// TwinCAT 3 PLC project PLC
// ProgramVersion: 3.1.4024.0
// libraries:
//   Tc2_Standard, * (Beckhoff Automation GmbH)
//   Tc2_System, * (Beckhoff Automation GmbH)
//   Tc2_Utilities, * (Beckhoff Automation GmbH)
//   Tc3_IotBase, * (Beckhoff Automation GmbH)
//   Tc3_IotCommunicator, * (Beckhoff Automation GmbH)
//   Tc3_Module, * (Beckhoff Automation GmbH)
// project tree:
//   00_HMI/DUTs/ ST_HMI_Variable_Mapping.TcDUT, ST_IoT_Device_General.TcDUT
//   00_HMI/DUTs/Widgets/ ST_IoT_HMI_General_Widget.TcDUT, ST_IoT_HMI_General_Widget_Plug.TcDUT, ST_IoT_HMI_General_Widget_RGBW.TcDUT, ST_IoT_HMI_General_Widget_Timer.TcDUT
//   DUTs/ProjectSpecific/HMI/00_Home/ ST_IoT_HMI_Rooms.TcDUT
//   DUTs/ProjectSpecific/HMI/100_FirstFloor/110_Entrance/ ST_IoT_HMI_Entrance.TcDUT
//   DUTs/ProjectSpecific/HMI/100_FirstFloor/120_Toilette/ ST_IoT_HMI_Toilette.TcDUT
//   DUTs/ProjectSpecific/HMI/100_FirstFloor/130_LivingRoom/ ST_IoT_HMI_LivingRoom.TcDUT
//   DUTs/ProjectSpecific/HMI/100_FirstFloor/140_Kitchen/ ST_IoT_HMI_Kitchen.TcDUT
//   DUTs/ProjectSpecific/HMI/100_FirstFloor/150_Storage/ ST_IoT_HMI_Storage.TcDUT
//   DUTs/ProjectSpecific/HMI/200_SecondFloor/210_Stairs/ ST_IoT_HMI_Stairs.TcDUT
//   DUTs/ProjectSpecific/HMI/200_SecondFloor/220_Office/ ST_IoT_HMI_Office.TcDUT
//   DUTs/ProjectSpecific/HMI/200_SecondFloor/230_Bathroom/ ST_IoT_HMI_Bathroom.TcDUT
//   DUTs/ProjectSpecific/HMI/200_SecondFloor/240_Bedroom/ ST_IoT_HMI_Bedroom.TcDUT
//   DUTs/ProjectSpecific/Rooms/Devices/ ST_Esp32_BedLight.TcDUT, ST_StatusDevices.TcDUT, ST_StatusShellyOnePM.TcDUT
//   DUTs/ProjectSpecific/Rooms/ ST_BedroomDevices.TcDUT, ST_LivingRoomDevices.TcDUT
//   / FC_MemcpyLimited.TcPOU, PlcTask.TcTTO
//   GVLs/ GVL_HMI.TcGVL, GVL_Devices.TcGVL
//   00_MQTT/DUT/ ST_MqttClient.TcDUT, ST_MqttConfig.TcDUT, ST_MqttData.TcDUT
//   00_MQTT/GVL/ GVL_Mqtt.TcGVL
//   POUs/00_HMI_Connection/ FB_IoT_HMI_Connection.TcPOU, PRG_IoT_HMI_Connection.TcPOU
//   POUs/00_MQTT_Connection/ FB_IoT_MqttClient.TcPOU
//   POUs/130_LivingRoom/ FB_LivingRoom.TcPOU, PRG_LivingRoom.TcPOU
//   POUs/ MAIN.TcPOU
// real-time tasks:
//   TASK PlcTask: cycle T#10ms, priority 6, ADS port 350

CONFIGURATION PLC
    RESOURCE PLC ON TwinCAT3
        TASK PlcTask(INTERVAL := T#10ms, PRIORITY := 6);
        PROGRAM MAIN WITH PlcTask : MAIN;
    END_RESOURCE
END_CONFIGURATION

// ---- 00_HMI/DUTs/ST_HMI_Variable_Mapping.TcDUT
TYPE ST_HMI_Variable_Mapping :
STRUCT
	sPath					: BOOL;
	
END_STRUCT
END_TYPE

// ---- 00_HMI/DUTs/ST_IoT_Device_General.TcDUT
TYPE ST_IoT_Device_General :
STRUCT

	sDeviceName					: STRING;	
	sDeviceIcon					: STRING;
	sMainTopic					: STRING;
	
END_STRUCT
END_TYPE

// ---- 00_HMI/DUTs/Widgets/ST_IoT_HMI_General_Widget.TcDUT
TYPE ST_IoT_HMI_General_Widget :
STRUCT
	sDisplayName 				: STRING := '';
	bValue1 					: BOOL := FALSE;
	{attribute 'iot.Unit' := '%'}
	{attribute 'iot.MinValue' := '0'}
	{attribute 'iot.MaxValue' := '100'}
	nValue2 					: INT;
	nValue2Request 				: INT;
	bValue2Up 					: BOOL;
	bValue2Down 				: BOOL;
	{attribute 'iot.Unit' := '%'}
	{attribute 'iot.MinValue' := '0'}
	{attribute 'iot.MaxValue' := '100'}
	nValue3 					: INT;
	nValue3Request 				: INT;
	bValue3Up 					: BOOL;
	bValue3Down 				: BOOL;
	sMode1 						: STRING := 'Automatic';
	aModes1 					: ARRAY[0..1] OF STRING := ['Manual', 'Automatic'];
	sMode2 						: STRING := 'Automatic';
	aModes2 					: ARRAY[0..2] OF STRING := ['Manual', 'Automatic', 'Next Mode'];
	sMode3 						: STRING := 'Automatic';
	aModes3 					: ARRAY[0..1] OF STRING := ['Manual', 'Automatic'];
END_STRUCT
END_TYPE

// ---- 00_HMI/DUTs/Widgets/ST_IoT_HMI_General_Widget_Plug.TcDUT
TYPE ST_IoT_HMI_General_Widget_Plug :
STRUCT
	
	sDisplayName 					: STRING := 'Plug';
	bOn 							: BOOL;
	sMode 							: STRING := 'Automatic';
	aModes 							: ARRAY[0..1] OF STRING := ['Manual', 'Automatic'];
	
END_STRUCT
END_TYPE

// ---- 00_HMI/DUTs/Widgets/ST_IoT_HMI_General_Widget_RGBW.TcDUT
TYPE ST_IoT_HMI_General_Widget_RGBW :
STRUCT
	sDisplayName 						: STRING := '';
	bLight 								: BOOL := FALSE;
	{attribute 'iot.Unit' := '%'}
	{attribute 'iot.MinValue' := '0'}
	{attribute 'iot.MaxValue' := '100'}
	nLight 								: INT := 100;
	nHueValue 							: INT := 57;
	nSaturation 						: INT := 100;
	{attribute 'iot.MinValue' := '2400'} 
	{attribute 'iot.MaxValue' := '6500'}
	nColorTemperature 					: INT := 3500;
	sMode 								: STRING := 'Permanent';
	aModes 								: ARRAY[0..4] OF STRING := ['Permanent', '15 Minuten', '30 Minuten', '45 Minuten', '1 Stunde'];
END_STRUCT
END_TYPE

// ---- 00_HMI/DUTs/Widgets/ST_IoT_HMI_General_Widget_Timer.TcDUT
TYPE ST_IoT_HMI_General_Widget_Timer :
STRUCT
	bLight			: BOOL;
	{attribute 'iot.Unit':='min'}
	{attribute 'iot.MinValue':='0'}
	{attribute 'iot.MaxValue':='120'}
	nLight			: INT;	
	sMode			: STRING;
	aModes			: ARRAY[0..1] OF STRING;
END_STRUCT
END_TYPE

// ---- DUTs/ProjectSpecific/HMI/00_Home/ST_IoT_HMI_Rooms.TcDUT
TYPE ST_IoT_HMI_Rooms :
STRUCT
	
	// First floor
	{attribute 'iot.DisplayName' := 'Flur UG'}
	{attribute 'iot.NestedStructIcon' := 'Door_Open'}
	sEntrance					: ST_IoT_HMI_Entrance;	
	{attribute 'iot.DisplayName' := 'Toilette'}
	{attribute 'iot.NestedStructIcon' := 'Toilet'}
	sToilette					: ST_IoT_HMI_Toilette;
	{attribute 'iot.DisplayName' := 'Wohnzimmer'}
	{attribute 'iot.NestedStructIcon' := 'Sofa'}
	sLivingRoom					: ST_IoT_HMI_LivingRoom;
	{attribute 'iot.DisplayName' := 'Kueche'}
	{attribute 'iot.NestedStructIcon' := 'Kitchen'}
	sKitchen					: ST_IoT_HMI_Kitchen;
	{attribute 'iot.DisplayName' := 'Speiss'}
	{attribute 'iot.NestedStructIcon' := 'Storage'}
	sStorage					: ST_IoT_HMI_Storage;
	
	// Second floor
	{attribute 'iot.DisplayName' := 'Flur OG'}
	{attribute 'iot.NestedStructIcon' := 'Floor'}
	sStairs						: ST_IoT_HMI_Stairs;
	{attribute 'iot.DisplayName' := 'Buero'}
	{attribute 'iot.NestedStructIcon' := 'PC'}
	sOffice						: ST_IoT_HMI_Office;
	{attribute 'iot.DisplayName' := 'Badezimmer'}
	{attribute 'iot.NestedStructIcon' := 'Bath'}
	sBathroom					: ST_IoT_HMI_Bathroom;
	{attribute 'iot.DisplayName' := 'Schlafzimmer'}
	{attribute 'iot.NestedStructIcon' := 'Bed'}
	sBedroom					: ST_IoT_HMI_Bedroom;
	
END_STRUCT
END_TYPE

// ---- DUTs/ProjectSpecific/HMI/100_FirstFloor/110_Entrance/ST_IoT_HMI_Entrance.TcDUT
TYPE ST_IoT_HMI_Entrance :
STRUCT
	
	{attribute 'iot.ReadOnly' := 'false'}
	{attribute 'iot.DisplayName' := 'Light'}
	{attribute 'iot.WidgetType' := 'General'}
	{attribute 'iot.GeneralWidgetIcon' := 'Lightbulb'}
	{attribute 'iot.GeneralWidgetColor' := 'LightSlateGray'}
	{attribute 'iot.GeneralValue1SwitchVisible' := 'true'}
	{attribute 'iot.GeneralValue2Visible' := 'false'}
	{attribute 'iot.GeneralValue2SliderVisible' := 'false'}
	{attribute 'iot.GeneralValue2SliderValuesVisible' := 'false'}
	{attribute 'iot.GeneralValue2SliderButtonsVisible' := 'false'}
	{attribute 'iot.GeneralValue2SliderButtonsInverted' := 'false'}
	{attribute 'iot.GeneralValue3Visible' := 'false'}
	{attribute 'iot.GeneralValue3SliderVisible' := 'false'}
	{attribute 'iot.GeneralValue3SliderValuesVisible' := 'false'}
	{attribute 'iot.GeneralValue3SliderButtonsVisible' := 'false'}
	{attribute 'iot.GeneralValue3SliderButtonsInverted' := 'false'}
	{attribute 'iot.GeneralMode1Visible' := 'false'}
	{attribute 'iot.GeneralMode1Changeable' := 'false'}
	{attribute 'iot.GeneralMode2Visible' := 'false'}
	{attribute 'iot.GeneralMode2Changeable' := 'false'}
	{attribute 'iot.GeneralMode3Visible' := 'false'}
	{attribute 'iot.GeneralMode3Changeable' := 'false'}
	sLight						: ST_IoT_HMI_General_Widget;
    
	{attribute 'iot.ReadOnly' := 'false'}
	{attribute 'iot.DisplayName' := 'Steckdose'}
	{attribute 'iot.WidgetType' := 'Plug'}
	{attribute 'iot.PlugModeVisible' := 'true'}
	{attribute 'iot.PlugModeChangeable' := 'true'}
	sPlug					 	: ST_IoT_HMI_General_Widget_Plug;		

END_STRUCT
END_TYPE

// ---- DUTs/ProjectSpecific/HMI/100_FirstFloor/120_Toilette/ST_IoT_HMI_Toilette.TcDUT
TYPE ST_IoT_HMI_Toilette :
STRUCT
	
	{attribute 'iot.ReadOnly' := 'false'}
	{attribute 'iot.DisplayName' := 'Light'}
	{attribute 'iot.WidgetType' := 'General'}
	{attribute 'iot.GeneralWidgetIcon' := 'Lightbulb'}
	{attribute 'iot.GeneralWidgetColor' := 'FF00BFFF'}
	{attribute 'iot.GeneralValue1SwitchVisible' := 'true'}
	{attribute 'iot.GeneralValue2Visible' := 'false'}
	{attribute 'iot.GeneralValue2SliderVisible' := 'false'}
	{attribute 'iot.GeneralValue2SliderValuesVisible' := 'false'}
	{attribute 'iot.GeneralValue2SliderButtonsVisible' := 'false'}
	{attribute 'iot.GeneralValue2SliderButtonsInverted' := 'false'}
	{attribute 'iot.GeneralValue3Visible' := 'false'}
	{attribute 'iot.GeneralValue3SliderVisible' := 'false'}
	{attribute 'iot.GeneralValue3SliderValuesVisible' := 'false'}
	{attribute 'iot.GeneralValue3SliderButtonsVisible' := 'false'}
	{attribute 'iot.GeneralValue3SliderButtonsInverted' := 'false'}
	{attribute 'iot.GeneralMode1Visible' := 'false'}
	{attribute 'iot.GeneralMode1Changeable' := 'false'}
	{attribute 'iot.GeneralMode2Visible' := 'false'}
	{attribute 'iot.GeneralMode2Changeable' := 'false'}
	{attribute 'iot.GeneralMode3Visible' := 'false'}
	{attribute 'iot.GeneralMode3Changeable' := 'false'}
	sLight						: ST_IoT_HMI_General_Widget;
    
	{attribute 'iot.ReadOnly' := 'false'}
	{attribute 'iot.DisplayName' := 'Steckdose'}
	{attribute 'iot.WidgetType' := 'Plug'}
	{attribute 'iot.PlugModeVisible' := 'true'}
	{attribute 'iot.PlugModeChangeable' := 'true'}
	sPlug					 	: ST_IoT_HMI_General_Widget_Plug;	

END_STRUCT
END_TYPE

// ---- DUTs/ProjectSpecific/HMI/100_FirstFloor/130_LivingRoom/ST_IoT_HMI_LivingRoom.TcDUT
TYPE ST_IoT_HMI_LivingRoom :
STRUCT
	
	{attribute 'iot.ReadOnly' := 'false'}
	{attribute 'iot.DisplayName' := 'Light'}
	{attribute 'iot.WidgetType' := 'General'}
	{attribute 'iot.GeneralWidgetIcon' := 'Lightbulb'}
	{attribute 'iot.GeneralWidgetColor' := 'FF00BFFF'}
	{attribute 'iot.GeneralValue1SwitchVisible' := 'true'}
	{attribute 'iot.GeneralValue2Visible' := 'false'}
	{attribute 'iot.GeneralValue2SliderVisible' := 'false'}
	{attribute 'iot.GeneralValue2SliderValuesVisible' := 'false'}
	{attribute 'iot.GeneralValue2SliderButtonsVisible' := 'false'}
	{attribute 'iot.GeneralValue2SliderButtonsInverted' := 'false'}
	{attribute 'iot.GeneralValue3Visible' := 'false'}
	{attribute 'iot.GeneralValue3SliderVisible' := 'false'}
	{attribute 'iot.GeneralValue3SliderValuesVisible' := 'false'}
	{attribute 'iot.GeneralValue3SliderButtonsVisible' := 'false'}
	{attribute 'iot.GeneralValue3SliderButtonsInverted' := 'false'}
	{attribute 'iot.GeneralMode1Visible' := 'false'}
	{attribute 'iot.GeneralMode1Changeable' := 'false'}
	{attribute 'iot.GeneralMode2Visible' := 'false'}
	{attribute 'iot.GeneralMode2Changeable' := 'false'}
	{attribute 'iot.GeneralMode3Visible' := 'false'}
	{attribute 'iot.GeneralMode3Changeable' := 'false'}
	sLight						: ST_IoT_HMI_General_Widget;
    
	{attribute 'iot.ReadOnly' := 'false'}
	{attribute 'iot.DisplayName' := 'Steckdose'}
	{attribute 'iot.WidgetType' := 'Plug'}
	{attribute 'iot.PlugModeVisible' := 'true'}
	{attribute 'iot.PlugModeChangeable' := 'true'}
	sPlug					 	: ST_IoT_HMI_General_Widget_Plug;	

END_STRUCT
END_TYPE

// ---- DUTs/ProjectSpecific/HMI/100_FirstFloor/140_Kitchen/ST_IoT_HMI_Kitchen.TcDUT
TYPE ST_IoT_HMI_Kitchen :
STRUCT
	
	{attribute 'iot.ReadOnly' := 'false'}
	{attribute 'iot.DisplayName' := 'Light'}
	{attribute 'iot.WidgetType' := 'General'}
	{attribute 'iot.GeneralWidgetIcon' := 'Lightbulb'}
	{attribute 'iot.GeneralWidgetColor' := 'FF00BFFF'}
	{attribute 'iot.GeneralValue1SwitchVisible' := 'true'}
	{attribute 'iot.GeneralValue2Visible' := 'false'}
	{attribute 'iot.GeneralValue2SliderVisible' := 'false'}
	{attribute 'iot.GeneralValue2SliderValuesVisible' := 'false'}
	{attribute 'iot.GeneralValue2SliderButtonsVisible' := 'false'}
	{attribute 'iot.GeneralValue2SliderButtonsInverted' := 'false'}
	{attribute 'iot.GeneralValue3Visible' := 'false'}
	{attribute 'iot.GeneralValue3SliderVisible' := 'false'}
	{attribute 'iot.GeneralValue3SliderValuesVisible' := 'false'}
	{attribute 'iot.GeneralValue3SliderButtonsVisible' := 'false'}
	{attribute 'iot.GeneralValue3SliderButtonsInverted' := 'false'}
	{attribute 'iot.GeneralMode1Visible' := 'false'}
	{attribute 'iot.GeneralMode1Changeable' := 'false'}
	{attribute 'iot.GeneralMode2Visible' := 'false'}
	{attribute 'iot.GeneralMode2Changeable' := 'false'}
	{attribute 'iot.GeneralMode3Visible' := 'false'}
	{attribute 'iot.GeneralMode3Changeable' := 'false'}
	sLight						: ST_IoT_HMI_General_Widget;
    
	{attribute 'iot.ReadOnly' := 'false'}
	{attribute 'iot.DisplayName' := 'Steckdose'}
	{attribute 'iot.WidgetType' := 'Plug'}
	{attribute 'iot.PlugModeVisible' := 'true'}
	{attribute 'iot.PlugModeChangeable' := 'true'}
	sPlug					 	: ST_IoT_HMI_General_Widget_Plug;	

END_STRUCT
END_TYPE

// ---- DUTs/ProjectSpecific/HMI/100_FirstFloor/150_Storage/ST_IoT_HMI_Storage.TcDUT
TYPE ST_IoT_HMI_Storage :
STRUCT
	
	{attribute 'iot.ReadOnly' := 'false'}
	{attribute 'iot.DisplayName' := 'Light'}
	{attribute 'iot.WidgetType' := 'General'}
	{attribute 'iot.GeneralWidgetIcon' := 'Lightbulb'}
	{attribute 'iot.GeneralWidgetColor' := 'FF00BFFF'}
	{attribute 'iot.GeneralValue1SwitchVisible' := 'true'}
	{attribute 'iot.GeneralValue2Visible' := 'false'}
	{attribute 'iot.GeneralValue2SliderVisible' := 'false'}
	{attribute 'iot.GeneralValue2SliderValuesVisible' := 'false'}
	{attribute 'iot.GeneralValue2SliderButtonsVisible' := 'false'}
	{attribute 'iot.GeneralValue2SliderButtonsInverted' := 'false'}
	{attribute 'iot.GeneralValue3Visible' := 'false'}
	{attribute 'iot.GeneralValue3SliderVisible' := 'false'}
	{attribute 'iot.GeneralValue3SliderValuesVisible' := 'false'}
	{attribute 'iot.GeneralValue3SliderButtonsVisible' := 'false'}
	{attribute 'iot.GeneralValue3SliderButtonsInverted' := 'false'}
	{attribute 'iot.GeneralMode1Visible' := 'false'}
	{attribute 'iot.GeneralMode1Changeable' := 'false'}
	{attribute 'iot.GeneralMode2Visible' := 'false'}
	{attribute 'iot.GeneralMode2Changeable' := 'false'}
	{attribute 'iot.GeneralMode3Visible' := 'false'}
	{attribute 'iot.GeneralMode3Changeable' := 'false'}
	sLight						: ST_IoT_HMI_General_Widget;
    
	{attribute 'iot.ReadOnly' := 'false'}
	{attribute 'iot.DisplayName' := 'Steckdose'}
	{attribute 'iot.WidgetType' := 'Plug'}
	{attribute 'iot.PlugModeVisible' := 'true'}
	{attribute 'iot.PlugModeChangeable' := 'true'}
	sPlug					 	: ST_IoT_HMI_General_Widget_Plug;	

END_STRUCT
END_TYPE

// ---- DUTs/ProjectSpecific/HMI/200_SecondFloor/210_Stairs/ST_IoT_HMI_Stairs.TcDUT
TYPE ST_IoT_HMI_Stairs :
STRUCT
	
	{attribute 'iot.ReadOnly' := 'false'}
	{attribute 'iot.DisplayName' := 'Light'}
	{attribute 'iot.WidgetType' := 'General'}
	{attribute 'iot.GeneralWidgetIcon' := 'Lightbulb'}
	{attribute 'iot.GeneralWidgetColor' := 'FF00BFFF'}
	{attribute 'iot.GeneralValue1SwitchVisible' := 'true'}
	{attribute 'iot.GeneralValue2Visible' := 'false'}
	{attribute 'iot.GeneralValue2SliderVisible' := 'false'}
	{attribute 'iot.GeneralValue2SliderValuesVisible' := 'false'}
	{attribute 'iot.GeneralValue2SliderButtonsVisible' := 'false'}
	{attribute 'iot.GeneralValue2SliderButtonsInverted' := 'false'}
	{attribute 'iot.GeneralValue3Visible' := 'false'}
	{attribute 'iot.GeneralValue3SliderVisible' := 'false'}
	{attribute 'iot.GeneralValue3SliderValuesVisible' := 'false'}
	{attribute 'iot.GeneralValue3SliderButtonsVisible' := 'false'}
	{attribute 'iot.GeneralValue3SliderButtonsInverted' := 'false'}
	{attribute 'iot.GeneralMode1Visible' := 'false'}
	{attribute 'iot.GeneralMode1Changeable' := 'false'}
	{attribute 'iot.GeneralMode2Visible' := 'false'}
	{attribute 'iot.GeneralMode2Changeable' := 'false'}
	{attribute 'iot.GeneralMode3Visible' := 'false'}
	{attribute 'iot.GeneralMode3Changeable' := 'false'}
	sLight						: ST_IoT_HMI_General_Widget;
    
	{attribute 'iot.ReadOnly' := 'false'}
	{attribute 'iot.DisplayName' := 'Steckdose'}
	{attribute 'iot.WidgetType' := 'Plug'}
	{attribute 'iot.PlugModeVisible' := 'true'}
	{attribute 'iot.PlugModeChangeable' := 'true'}
	sPlug					 	: ST_IoT_HMI_General_Widget_Plug;	

END_STRUCT
END_TYPE

// ---- DUTs/ProjectSpecific/HMI/200_SecondFloor/220_Office/ST_IoT_HMI_Office.TcDUT
TYPE ST_IoT_HMI_Office :
STRUCT
	
	{attribute 'iot.ReadOnly' := 'false'}
	{attribute 'iot.DisplayName' := 'Light'}
	{attribute 'iot.WidgetType' := 'General'}
	{attribute 'iot.GeneralWidgetIcon' := 'Lightbulb'}
	{attribute 'iot.GeneralWidgetColor' := 'FF00BFFF'}
	{attribute 'iot.GeneralValue1SwitchVisible' := 'true'}
	{attribute 'iot.GeneralValue2Visible' := 'false'}
	{attribute 'iot.GeneralValue2SliderVisible' := 'false'}
	{attribute 'iot.GeneralValue2SliderValuesVisible' := 'false'}
	{attribute 'iot.GeneralValue2SliderButtonsVisible' := 'false'}
	{attribute 'iot.GeneralValue2SliderButtonsInverted' := 'false'}
	{attribute 'iot.GeneralValue3Visible' := 'false'}
	{attribute 'iot.GeneralValue3SliderVisible' := 'false'}
	{attribute 'iot.GeneralValue3SliderValuesVisible' := 'false'}
	{attribute 'iot.GeneralValue3SliderButtonsVisible' := 'false'}
	{attribute 'iot.GeneralValue3SliderButtonsInverted' := 'false'}
	{attribute 'iot.GeneralMode1Visible' := 'false'}
	{attribute 'iot.GeneralMode1Changeable' := 'false'}
	{attribute 'iot.GeneralMode2Visible' := 'false'}
	{attribute 'iot.GeneralMode2Changeable' := 'false'}
	{attribute 'iot.GeneralMode3Visible' := 'false'}
	{attribute 'iot.GeneralMode3Changeable' := 'false'}
	sLight						: ST_IoT_HMI_General_Widget;
    
	{attribute 'iot.ReadOnly' := 'false'}
	{attribute 'iot.DisplayName' := 'Steckdose'}
	{attribute 'iot.WidgetType' := 'Plug'}
	{attribute 'iot.PlugModeVisible' := 'true'}
	{attribute 'iot.PlugModeChangeable' := 'true'}
	sPlug					 	: ST_IoT_HMI_General_Widget_Plug;	

END_STRUCT
END_TYPE

// ---- DUTs/ProjectSpecific/HMI/200_SecondFloor/230_Bathroom/ST_IoT_HMI_Bathroom.TcDUT
TYPE ST_IoT_HMI_Bathroom :
STRUCT
	
	{attribute 'iot.ReadOnly' := 'false'}
	{attribute 'iot.DisplayName' := 'Light'}
	{attribute 'iot.WidgetType' := 'General'}
	{attribute 'iot.GeneralWidgetIcon' := 'Lightbulb'}
	{attribute 'iot.GeneralWidgetColor' := 'FF00BFFF'}
	{attribute 'iot.GeneralValue1SwitchVisible' := 'true'}
	{attribute 'iot.GeneralValue2Visible' := 'false'}
	{attribute 'iot.GeneralValue2SliderVisible' := 'false'}
	{attribute 'iot.GeneralValue2SliderValuesVisible' := 'false'}
	{attribute 'iot.GeneralValue2SliderButtonsVisible' := 'false'}
	{attribute 'iot.GeneralValue2SliderButtonsInverted' := 'false'}
	{attribute 'iot.GeneralValue3Visible' := 'false'}
	{attribute 'iot.GeneralValue3SliderVisible' := 'false'}
	{attribute 'iot.GeneralValue3SliderValuesVisible' := 'false'}
	{attribute 'iot.GeneralValue3SliderButtonsVisible' := 'false'}
	{attribute 'iot.GeneralValue3SliderButtonsInverted' := 'false'}
	{attribute 'iot.GeneralMode1Visible' := 'false'}
	{attribute 'iot.GeneralMode1Changeable' := 'false'}
	{attribute 'iot.GeneralMode2Visible' := 'false'}
	{attribute 'iot.GeneralMode2Changeable' := 'false'}
	{attribute 'iot.GeneralMode3Visible' := 'false'}
	{attribute 'iot.GeneralMode3Changeable' := 'false'}
	sLight						: ST_IoT_HMI_General_Widget;
    
	{attribute 'iot.ReadOnly' := 'false'}
	{attribute 'iot.DisplayName' := 'Steckdose'}
	{attribute 'iot.WidgetType' := 'Plug'}
	{attribute 'iot.PlugModeVisible' := 'true'}
	{attribute 'iot.PlugModeChangeable' := 'true'}
	sPlug					 	: ST_IoT_HMI_General_Widget_Plug;	

END_STRUCT
END_TYPE

// ---- DUTs/ProjectSpecific/HMI/200_SecondFloor/240_Bedroom/ST_IoT_HMI_Bedroom.TcDUT
TYPE ST_IoT_HMI_Bedroom :
STRUCT
	
	{attribute 'iot.ReadOnly' := 'false'}
	{attribute 'iot.DisplayName' := 'Bett Licht'}
	{attribute 'iot.WidgetType' := 'RGBW'}
	{attribute 'iot.LightValueVisible' := 'true'}
	{attribute 'iot.LightSliderVisible' := 'true'}
	{attribute 'iot.LightColorPaletteVisible' := 'true'}
	{attribute 'iot.LightColorTemperatureSliderVisible' := 'false'}
	{attribute 'iot.LightModeVisible' := 'true'}
	{attribute 'iot.LightModeChangeable' := 'true'}
	sEsp32_BedLight			 : ST_IoT_HMI_General_Widget_RGBW;

END_STRUCT
END_TYPE

// ---- DUTs/ProjectSpecific/Rooms/Devices/ST_Esp32_BedLight.TcDUT
TYPE ST_Esp32_BedLight :
STRUCT

	xOn					: BOOL;
	stMode				: STRING;

	iRed				: INT;
	iGreen				: INT;
	iBlue				: INT;	

END_STRUCT
END_TYPE

// ---- DUTs/ProjectSpecific/Rooms/Devices/ST_StatusDevices.TcDUT
TYPE ST_StatusDevices :
STRUCT

	sLivingRoom						: ST_LivingRoomDevices;
	sBedroom						: ST_BedroomDevices;

END_STRUCT
END_TYPE

// ---- DUTs/ProjectSpecific/Rooms/Devices/ST_StatusShellyOnePM.TcDUT
TYPE ST_StatusShellyOnePM :
STRUCT

	iOutput					: INT; // -1..status not set, 0..output = false, 1..output = true	

END_STRUCT
END_TYPE

// ---- DUTs/ProjectSpecific/Rooms/ST_BedroomDevices.TcDUT
TYPE ST_BedroomDevices :
STRUCT

	sEsp32_BedLight						: ST_Esp32_BedLight;	

END_STRUCT
END_TYPE

// ---- DUTs/ProjectSpecific/Rooms/ST_LivingRoomDevices.TcDUT
TYPE ST_LivingRoomDevices :
STRUCT

	sShellyLight						: ST_StatusShellyOnePM;	
	
END_STRUCT
END_TYPE

// ---- 00_MQTT/DUT/ST_MqttClient.TcDUT
TYPE ST_MqttClient :
STRUCT

	sConfig				: st_MqttConfig;	

	fbIotMqttClient		: FB_IoT_MqttClient;

	sData				: ST_MqttData;
	
END_STRUCT
END_TYPE

// ---- 00_MQTT/DUT/ST_MqttConfig.TcDUT
TYPE ST_MqttConfig :
STRUCT
	
	xEnable						: BOOL := FALSE;
	sHostName 					: STRING := 'localhost';
    nHostPort 					: UINT := 1883;
	
END_STRUCT
END_TYPE

// ---- 00_MQTT/DUT/ST_MqttData.TcDUT
TYPE ST_MqttData :
STRUCT
	
	stTopic					: STRING(255);
	stMessage				: STRING(255);

END_STRUCT
END_TYPE

// ---- GVLs/GVL_HMI.TcGVL
{attribute 'qualified_only'}
VAR_GLOBAL

	sDevice					: ST_IoT_Device_General;
	sRooms					: ST_IoT_HMI_Rooms;

END_VAR

// ---- GVLs/GVL_Devices.TcGVL
{attribute 'qualified_only'}
VAR_GLOBAL

	sStatus					: ST_StatusDevices;

END_VAR

// ---- 00_MQTT/GVL/GVL_Mqtt.TcGVL
{attribute 'qualified_only'}
VAR_GLOBAL

	sClient						: ST_MqttClient;	

END_VAR

// ---- POUs/MAIN.TcPOU
PROGRAM MAIN
VAR
END_VAR


	 
PRG_LivingRoom();

PRG_IoT_HMI_Connection();

END_PROGRAM

// ---- POUs/130_LivingRoom/PRG_LivingRoom.TcPOU
PROGRAM PRG_LivingRoom
VAR_INPUT
END_VAR
VAR_OUTPUT
END_VAR
VAR
	fbLivingRoom					: FB_LivingRoom;
END_VAR

(*
****************************************************************************************************************************

****************************************************************************************************************************

Erstellt:       FÖB      20.09.2022
 
Geändert:       

****************************************************************************************************************************
Was man wissen sollte:

****************************************************************************************************************************
*)

//**************************************************************************************************************************
// Aufruf Ablaufsteuerung
//**************************************************************************************************************************

fbLivingRoom(
	ixErrorAcknowledge:= , 
	ixAcknowledgePulse:= , 
	sHmi:= GVL_HMI.sRooms.sLivingRoom, 
	sMqttClient:= GVL_Mqtt.sClient, 
	sStatusDevices:= GVL_Devices.sStatus);

END_PROGRAM

// ---- POUs/130_LivingRoom/FB_LivingRoom.TcPOU
FUNCTION_BLOCK FB_LivingRoom

VAR_INPUT
	
	ixErrorAcknowledge 							: BOOL;                 
	ixAcknowledgePulse 							: BOOL;      
	
END_VAR                             			
                                    			
VAR_IN_OUT     
	
	//================================================================================
	// HMI interface
	sHmi										: ST_IoT_HMI_LivingRoom;
	
	//================================================================================
	// MQTT data
	sMqttClient									: ST_MqttClient;
	
	//================================================================================
	// MQTT data
	sStatusDevices								: ST_StatusDevices;
	
END_VAR                             			
                                    			
VAR_OUTPUT	 

	//================================================================================
	// Alarms       
	oxF_TestDeactivated 						: BOOL := TRUE; // Test is deactivated
	oxF_InterceptionCircuitTriggered 			: BOOL := TRUE; // Interception circuit has been triggered - please acknowledge                                                     
	oxF_InfeedStroke_HP							: BOOL := TRUE; // Infeed stroke does not reach home position
	oxF_InfeedStroke_WP							: BOOL := TRUE; // Infeed stroke does not reach working position 
    oxF_InfeedStroke_Pl							: BOOL := TRUE; // Infeed stroke plausibility		
	oxF_LiftingCyl_HP							: BOOL := TRUE; // Lifting cylinder does not reach home position
	oxF_LiftingCyl_WP							: BOOL := TRUE; // Lifting cylinder does not reach working position 
    oxF_LiftingCyl_Pl							: BOOL := TRUE; // Lifting cylinder plausibility                                                
	oxF_Wenglor_1_LimaServerNotConnected		: BOOL := TRUE; // Wenglor 1 - no connection to LIMA server
	oxF_Wenglor_1_ResultServerNotConnected		: BOOL := TRUE; // Wenglor 1 - no connection to result server
	oxF_Wenglor_1_ErrorRequestProjectLoad		: BOOL := TRUE; // Wenglor 1 - error during LIMA command "Project_Load"
	oxF_Wenglor_1_ErrorRequestDeviceTrigger		: BOOL := TRUE; // Wenglor 1 - error during LIMA command "Device_Trigger" 
	oxF_Wenglor_1_ResponseResultServer			: BOOL := TRUE; // Wenglor 1 - no response from result server                                            
	oxF_Wenglor_2_LimaServerNotConnected		: BOOL := TRUE; // Wenglor 2 - no connection to LIMA server
	oxF_Wenglor_2_ResultServerNotConnected		: BOOL := TRUE; // Wenglor 2 - no connection to result server
	oxF_Wenglor_2_ErrorRequestProjectLoad		: BOOL := TRUE; // Wenglor 2 - error during LIMA command "Project_Load"
	oxF_Wenglor_2_ErrorRequestDeviceTrigger		: BOOL := TRUE; // Wenglor 2 - error during LIMA command "Device_Trigger" 
	oxF_Wenglor_2_ResponseResultServer			: BOOL := TRUE; // Wenglor 2 - no response from result server
	oxF_LimaServerManuallyDisconnected			: BOOL := TRUE; // Wenglor - LIMA server manually disconnected
	oxF_CS_LogError								: BOOL := TRUE; // Control station error at Log command

END_VAR                                 		        
                                        		
VAR PERSISTENT    
                          		
	lxMessage 									: BOOL;
	lxOpModeOk									: BOOL;				 
	                                			
	lEdge_TippOk 								: R_TRIG;
	
	stStatusText								: STRING(255);
                                    			
	lxEntryAction 								: BOOL;
	lxStopped 									: BOOL;
	liStep 										: INT;
	liLStep 									: INT;
	liNStep 									: INT;
	liLastCycleStep 							: INT;
	liCounter_i 								: INT;
	liCounter_j 								: INT;
	              
	lxTonStep_IN 								: BOOL;
	lxTonStepF_IN 								: BOOL;
	ltTonStep_PT 								: TIME;
	ltTonStepF_PT 								: TIME;
	lTonStep 									: TON;
	lTonStepF 									: TON;

	//================================================================================
	// General

	//================================================================================
	// local HMI data

	//================================================================================
	// MQTT client	
	lstTopicPub									: STRING(255) := 'shellyplus1pm-e465b8944d64/command/switch:0';
	lstMessagePub								: STRING(255);
	lxPublish									: BOOL;
	lxPublished									: BOOL;
                               			
	lstTopicSub									: STRING(255) := 'shellyplus1pm-e465b8944d64/status/switch:0/#';
	lxSubscribed								: BOOL;
	lxUnsubscribed								: BOOL;
	
	//================================================================================
	// Get status of shelly device
	lTonStatusUpdate							: TON;
	lxTonStatusUpdate_IN						: BOOL;
	ltTonStatusUpdate_PT						: TIME;
	lxEnableGetStatus							: BOOL;
	lstStatusMessage							: STRING(255);
	
	lxRefreshDeviceStatus						: BOOL;
	
	//================================================================================  
	// Start Acess & Process required for Shelly
	lRE_StartAcess			     				: R_TRIG;
	lFE_StartAcess			     				: F_TRIG;
	lxProcessingRequired						: BOOL;
	lxStartAccess								: BOOL;

END_VAR

VAR_TEMP
	
END_VAR

VAR CONSTANT 
END_VAR

{region information}
(*
****************************************************************************************************************************
Living room
****************************************************************************************************************************

****************************************************************************************************************************
version history:

date            name        comment
10.10.2023      FÖB         creation

****************************************************************************************************************************
description:


****************************************************************************************************************************
*)
{endregion} 
//**************************************************************************************************************************
			

//**************************************************************************************************************************
{region mqtt client}

	sMqttClient.fbIotMqttClient(
			 					ixEnable := sMqttClient.sConfig.xEnable,
								sHostName := sMqttClient.sConfig.sHostName,
								nHostPort := sMqttClient.sConfig.nHostPort,
								sMqttData := sMqttClient.sData,
								sStatusDevices := sStatusDevices
								);

{endregion}

//**************************************************************************************************************************				 
{region reset}
		  
	IF NOT(sMqttClient.fbIotMqttClient.bConnected) OR  
		FALSE THEN

		lxEntryAction := TRUE;
		
		liLStep := liStep;
		liStep := 0;
	END_IF
		 
{endregion}

//**************************************************************************************************************************
{region error acknowledge}

	IF ixErrorAcknowledge THEN
		;	
	END_IF	

{endregion}

//**************************************************************************************************************************
{region check start access for indexer}
	
	lRE_StartAcess(CLK := sHmi.sLight.bValue1);
	lFE_StartAcess(CLK := sHmi.sLight.bValue1);
		 
	IF lRE_StartAcess.Q OR lFE_StartAcess.Q THEN

		//processing required through part tracking? 
		lxProcessingRequired := NOT(lxRefreshDeviceStatus);

		lxStartAccess := lxProcessingRequired;
	END_IF
	 
{endregion}

//**************************************************************************************************************************
{region state machine}
	
	CASE liStep OF
			
			//**************************************************************************************************************************
			// STEP 0
		0:
			lxStopped := TRUE;
				 
			lxMessage := TRUE;
			
			IF lxOpModeOk AND sMqttClient.fbIotMqttClient.bConnected THEN

				liStep := 2;
			END_IF

			//**************************************************************************************************************************
			// STEP 2
		2:
			IF lxEntryAction THEN
				lxEntryAction := FALSE;
			END_IF

			lxMessage := TRUE;
			
			IF lxOpModeOk THEN
	
		 		liStep := 10;
		 		IF lxSubscribed THEN
					liStep := 4; 
				END_IF
			END_IF

			//**************************************************************************************************************************
			// STEP 4 - unsubscribe topic
		4:
			IF lxEntryAction THEN
				lxEntryAction := FALSE;
			END_IF
		
			lxUnsubscribed := sMqttClient.fbIotMqttClient.Unsubscribe(lstTopicSub);

			IF NOT(lxUnsubscribed) THEN
				// StatusText:  '0--------1---------2---------3---------4---------5'
				stStatusText := 'Wait until topic unsubscribed';
			ELSE
				lxMessage := TRUE;
			END_IF
	
			IF lxUnsubscribed THEN
					 
				lxSubscribed := FALSE;
							   
				liStep := 10000;
			END_IF
				 
			//**************************************************************************************************************************
			// STEP 10 - Check if Log is pending
		10:
			IF lxEntryAction THEN
				lxEntryAction := FALSE;
			END_IF
		
			lxSubscribed := sMqttClient.fbIotMqttClient.Subscribe(lstTopicSub, TcIotMqttQos.AtMostOnceDelivery);

			IF NOT(lxSubscribed) THEN
				// StatusText:  '0--------1---------2---------3---------4---------5'
				stStatusText := 'Wait until topic subscribed';
			ELSE
				lxMessage := TRUE;
			END_IF
	
			IF lxSubscribed THEN

				liStep := 20;
			END_IF


			//**************************************************************************************************************************      
			//**************************************************************************************************************************      
			// STEP 20
			//**************************************************************************************************************************    
		20:
			IF lxEntryAction THEN
				lxEntryAction := FALSE;
			END_IF
			
			IF NOT (lxStartAccess) THEN
				// StatusText:  '0--------1---------2---------3---------4---------5'
				stStatusText := 'Wait for start access';
			ELSE
				lxMessage := TRUE;
			END_IF
				 
			lxStopped := NOT(lxStartAccess);

	 		lxTonStatusUpdate_IN := TRUE;
			ltTonStatusUpdate_PT := T#5S;
		  
			IF lxOpModeOk AND lxStartAccess THEN
				
				liStep := 100;
			ELSIF lTonStatusUpdate.Q THEN
						  
	 			liStep := 32000;	 
			END_IF	

	  
			//**************************************************************************************************************************        
			//**************************************************************************************************************************          
			// STEP 100 - Publish "toggle output"
		100:	
			IF lxEntryAction THEN
	 
				lxEntryAction := FALSE;
			END_IF	
											 
			lstMessagePub := 'toggle';				
			lxPublished := sMqttClient.fbIotMqttClient.Publish(sTopic:= lstTopicPub,
								pPayload:= ADR(lstMessagePub), 
								nPayloadSize:= LEN2(ADR(lstMessagePub)),
								eQoS:= TcIotMqttQos.AtMostOnceDelivery, 
								bRetain:= FALSE,
								bQueue := FALSE );
			
			IF NOT (lxPublished) THEN
				// StatusText:  '0--------1---------2---------3---------4---------5'
				stStatusText := 'Wait until message published';
			ELSE
				lxMessage := TRUE;
			END_IF
	
			IF lxPublished THEN

	 			lxStartAccess := FALSE;
		  
				liStep := 110;
			END_IF	 
     
			//**************************************************************************************************************************          
			// STEP 210 - Publish "toggle output"
		110:	
			IF lxEntryAction THEN
	 
				lxEntryAction := FALSE;
			END_IF	

			lxMessage := TRUE;
	
		 	lxTonStep_IN := TRUE;
			ltTonStep_PT := T#1S;
			  
			IF lTonStep.Q THEN
		  
				liStep := 32000;
			END_IF	

	 
			//**************************************************************************************************************************        
			//**************************************************************************************************************************          
			// STEP 32000 - Publish "status update"
		 32000:
			IF lxEntryAction THEN
					 
				sStatusDevices.sLivingRoom.sShellyLight.iOutput := -1;	
 
				lxEntryAction := FALSE;
			END_IF
 
	  
			lstMessagePub := 'status_update';				
			lxPublished := sMqttClient.fbIotMqttClient.Publish(sTopic:= lstTopicPub,
								pPayload:= ADR(lstMessagePub), 
								nPayloadSize:= LEN2(ADR(lstMessagePub)),
								eQoS:= TcIotMqttQos.AtMostOnceDelivery, 
								bRetain:= FALSE,
								bQueue := FALSE );
			
			IF NOT (lxPublished) THEN
				// StatusText:  '0--------1---------2---------3---------4---------5'
				stStatusText := 'Wait until message published';
			ELSE
				lxMessage := TRUE;
			END_IF
	
			IF lxPublished THEN
				liStep := 32010;
			END_IF
		    
			//**************************************************************************************************************************          
			// STEP 32010 - Publish "status update"
		32010:	
			IF lxEntryAction THEN
						  
				lxEntryAction := FALSE;
			END_IF
			
			IF (sStatusDevices.sLivingRoom.sShellyLight.iOutput = -1) THEN
				// StatusText:  '0--------1---------2---------3---------4---------5'
				stStatusText := 'Wait for data ready';
			ELSE
				lxMessage := TRUE;
			END_IF

			// Write status to HMI
			IF (sStatusDevices.sLivingRoom.sShellyLight.iOutput <> -1) THEN
				
				IF (sStatusDevices.sLivingRoom.sShellyLight.iOutput = 1) THEN		  
					sHmi.sLight.bValue1 := TRUE;
				ELSIF (sStatusDevices.sLivingRoom.sShellyLight.iOutput = 0) THEN		  
					sHmi.sLight.bValue1 := FALSE;
				END_IF
					 
				liStep := 32020;
			END_IF
		    
			//**************************************************************************************************************************          
			// STEP 32020 - Publish "status update"
		32020:	
			IF lxEntryAction THEN
						  
				lxEntryAction := FALSE;
			END_IF
			
			lxMessage := TRUE;

	 		lxTonStep_IN := TRUE;
			ltTonStep_PT := T#50MS;
		  
			IF lTonStep.Q THEN
					 
				liStep := 20;
			END_IF					 
	END_CASE
		 
{endregion}

//**************************************************************************************************************************
{region write status to hmi}
		 		  				
	lxRefreshDeviceStatus := (liStep >= 32000) AND (liStep < 32100);
			  
{endregion}
	
//**************************************************************************************************************************
{region error-monitoring}
	
	ErrorMonitoring();

{endregion}

//**************************************************************************************************************************
{region stepchain monitoring}

	StepchainMonitoring();

{endregion}

METHOD PRIVATE ErrorMonitoring : BOOL
//**************************************************************************************************************************
{region ERROR-MONITORING}
	
	

{endregion}
END_METHOD

{warning 'Methodenimplementierung hinzufügen'}
METHOD PRIVATE StepchainMonitoring : BOOL
//**************************************************************************************************************************
{region STEPCHAIN STEP MONITORING}
	
	IF liStep <> liLastCycleStep THEN
		lxEntryAction := TRUE;
		
		lxTonStep_IN := FALSE;
		lxTonStepF_IN := FALSE;
		lxTonStatusUpdate_IN := FALSE;
		
		liLStep := liLastCycleStep;
	END_IF
	liLastCycleStep := liStep;
	
{endregion}

//**************************************************************************************************************************
{region timer call}
	
	lTonStep(IN := lxTonStep_IN,
				 PT := ltTonStep_PT);
	lTonStepF(IN := lxTonStepF_IN,
				  PT := ltTonStepF_PT);
	lTonStatusUpdate(IN := lxTonStatusUpdate_IN,
				  PT := ltTonStatusUpdate_PT);
	
{endregion}
END_METHOD

END_FUNCTION_BLOCK

// ---- POUs/00_HMI_Connection/PRG_IoT_HMI_Connection.TcPOU
PROGRAM PRG_IoT_HMI_Connection
VAR_INPUT
END_VAR
VAR_OUTPUT
END_VAR
VAR
	fbIoT_HMI_Connection				: FB_IoT_HMI_Connection;
END_VAR

(*
****************************************************************************************************************************

****************************************************************************************************************************

Erstellt:       FÖB      20.09.2022
 
Geändert:       

****************************************************************************************************************************
Was man wissen sollte:

****************************************************************************************************************************
*)

//**************************************************************************************************************************
// Set device settings
GVL_HMI.sDevice.sDeviceName := 'Zuhause';
GVL_HMI.sDevice.sDeviceIcon := 'House';
GVL_HMI.sDevice.sMainTopic := 'home';

//**************************************************************************************************************************
// Aufruf Ablaufsteuerung
//**************************************************************************************************************************

fbIoT_HMI_Connection(
					sDeviceSettings:= GVL_HMI.sDevice, 
					sHMI:= GVL_HMI.sRooms
					);

END_PROGRAM

// ---- POUs/00_HMI_Connection/FB_IoT_HMI_Connection.TcPOU
FUNCTION_BLOCK FB_IoT_HMI_Connection
VAR_INPUT
END_VAR
VAR_IN_OUT
	sDeviceSettings					: ST_IoT_Device_General;
	sHmi							: ST_IoT_HMI_Rooms;
END_VAR
VAR_OUTPUT
END_VAR
VAR
	
	// Communicator function block with usage of SendData method
	fbIoT_HMI						: FB_IotCommunicator := ();
	
	lxHmiError						: BOOL;
	lhrHmiErrorCode					: HRESULT;
	//leConnectionState				: ;
	lxHmiConnected					: BOOL;
	
	lTonSendHmiData_IN				: BOOL;
	lTonSendHmiData	 				: TON;	
	
END_VAR

//**************************************************************************************************************************
// IoT HMI Communication

{region IoT HMI Communication}

	fbIoT_HMI.sHostName := '127.0.0.1';
	fbIoT_HMI.nPort := 1883;
	fbIoT_HMI.sMainTopic := sDeviceSettings.sMainTopic;
	fbIoT_HMI.sDevicename := sDeviceSettings.sDeviceName;
	fbIoT_HMI.sDeviceIcon := sDeviceSettings.sDeviceIcon;
	   
	lxHmiError := fbIoT_HMI.bError;
	lhrHmiErrorCode := fbIoT_HMI.hrErrorCode;
	//leHmiConnectionState := fbIoT_HMI.eConnectionState; 
	lxHmiConnected := fbIoT_HMI.bConnected;
	
	// Start executing IoT HMI			   
	fbIoT_HMI.Execute(TRUE);
	
	lTonSendHmiData_IN := lxHmiConnected;
		  
	IF lTonSendHmiData.Q THEN
		lTonSendHmiData_IN := FALSE;
					   
		fbIoT_HMI.SendData(ADR(sHMI),SIZEOF(sHMI));
	END_IF
		 
	lTonSendHmiData(IN := lTonSendHmiData_IN,
			 		PT := T#500MS);
		 
{endregion}


//**************************************************************************************************************************
// Get inputs from HMI

{region Get inputs from HMI}

	GetInputsFromHMI();

{endregion}

METHOD GetInputsFromHMI : BOOL
VAR_INPUT
END_VAR
IF fbIoT_HMI.fbCommand.bAvailable THEN
	
	// Entrance
	IF FALSE THEN
		;
	// Toilette
	ELSIF FALSE THEN
		;	
	// Living room
	ELSIF fbIoT_HMI.fbCommand.sVarName = 'sLivingRoom.sLight.bValue1' THEN
		fbIoT_HMI.fbCommand.GetValue(ADR(sHMI.sLivingRoom.sLight.bValue1), SIZEOF(sHMI.sLivingRoom.sLight.bValue1), E_IotCommunicatorDatatype.type_BOOL);
	ELSIF fbIoT_HMI.fbCommand.sVarName = 'sLivingRoom.sPlug.bOn' THEN
		fbIoT_HMI.fbCommand.GetValue(ADR(sHMI.sLivingRoom.sPlug.bOn), SIZEOF(sHMI.sLivingRoom.sPlug.bOn), E_IotCommunicatorDatatype.type_BOOL);
	ELSIF fbIoT_HMI.fbCommand.sVarName = 'sLivingRoom.sPlug.sMode' THEN
		fbIoT_HMI.fbCommand.GetValue(ADR(sHMI.sLivingRoom.sPlug.sMode), SIZEOF(sHMI.sLivingRoom.sPlug.sMode), E_IotCommunicatorDatatype.type_STRING);
	// Kitchen
	ELSIF FALSE THEN
		;	
	// Storage
	ELSIF FALSE THEN
		;	
	// Stairs
	ELSIF FALSE THEN
		;	
	// Office
	ELSIF FALSE THEN
		;	
	// Bathroom
	ELSIF FALSE THEN
		;	
	// Bedroom
	ELSIF fbIoT_HMI.fbCommand.sVarName = 'sBedroom.sEsp32_BedLight.bLight' THEN
		fbIoT_HMI.fbCommand.GetValue(ADR(sHMI.sBedroom.sEsp32_BedLight.bLight), SIZEOF(sHMI.sBedroom.sEsp32_BedLight.bLight), E_IotCommunicatorDatatype.type_BOOL);
	ELSIF fbIoT_HMI.fbCommand.sVarName = 'sBedroom.sEsp32_BedLight.nLight' THEN
		fbIoT_HMI.fbCommand.GetValue(ADR(sHMI.sBedroom.sEsp32_BedLight.nLight), SIZEOF(sHMI.sBedroom.sEsp32_BedLight.nLight), E_IotCommunicatorDatatype.type_INT);
	ELSIF fbIoT_HMI.fbCommand.sVarName = 'sBedroom.sEsp32_BedLight.nHueValue' THEN
		fbIoT_HMI.fbCommand.GetValue(ADR(sHMI.sBedroom.sEsp32_BedLight.nHueValue), SIZEOF(sHMI.sBedroom.sEsp32_BedLight.nHueValue), E_IotCommunicatorDatatype.type_INT);
	ELSIF fbIoT_HMI.fbCommand.sVarName = 'sBedroom.sEsp32_BedLight.nSaturation' THEN
		fbIoT_HMI.fbCommand.GetValue(ADR(sHMI.sBedroom.sEsp32_BedLight.nSaturation), SIZEOF(sHMI.sBedroom.sEsp32_BedLight.nSaturation), E_IotCommunicatorDatatype.type_INT);
	ELSIF fbIoT_HMI.fbCommand.sVarName = 'sBedroom.sEsp32_BedLight.nColorTemperature' THEN
		fbIoT_HMI.fbCommand.GetValue(ADR(sHMI.sBedroom.sEsp32_BedLight.nColorTemperature), SIZEOF(sHMI.sBedroom.sEsp32_BedLight.nColorTemperature), E_IotCommunicatorDatatype.type_INT);
	ELSIF fbIoT_HMI.fbCommand.sVarName = 'sBedroom.sEsp32_BedLight.sMode' THEN
		fbIoT_HMI.fbCommand.GetValue(ADR(sHMI.sBedroom.sEsp32_BedLight.sMode), SIZEOF(sHMI.sBedroom.sEsp32_BedLight.sMode), E_IotCommunicatorDatatype.type_STRING);
	ELSE
		// RETURN;
	END_IF	
	fbIoT_HMI.SendData(ADR(sHMI), SIZEOF(sHMI));
	fbIoT_HMI.fbCommand.Remove();
END_IF
END_METHOD

END_FUNCTION_BLOCK

// ---- FC_MemcpyLimited.TcPOU
FUNCTION FC_MemcpyLimited : BOOL
VAR_INPUT
	DestinationAdress			: PVOID;
	ediSizeOfDestAdress			: UDINT;
	
	SourceAdress				: PVOID;
	ediBytesToCopy				: UDINT;
END_VAR
VAR
	tdiBytesToCopy				: UDINT;
END_VAR

tdiBytesToCopy := LIMIT(0, ediBytesToCopy, ediSizeOfDestAdress);

MEMCPY(DestinationAdress, SourceAdress, tdiBytesToCopy);

END_FUNCTION

// ---- POUs/00_MQTT_Connection/FB_IoT_MqttClient.TcPOU
{attribute 'c++_compatible'}
FUNCTION_BLOCK FB_IoT_MqttClient EXTENDS FB_IotMqttClient
VAR_INPUT
	ixEnable						: BOOL;
END_VAR
VAR_IN_OUT

	sMqttData						: ST_MqttData;
	sStatusDevices					: ST_StatusDevices;	

END_VAR
VAR_OUTPUT
END_VAR
VAR	
END_VAR

Execute(ixEnable);

{attribute 'c++_compatible'}
{attribute 'pack_mode' := '4'}
{attribute 'show'}
{attribute 'minimal_input_size' := '4'}
METHOD OnMqttMessage : HRESULT
VAR_IN_OUT CONSTANT
topic 						: STRING;
END_VAR
VAR_INPUT
payload 					: PVOID;
length 						: UDINT;
qos 						: TcIotMqttQos;
repeated 					: BOOL;
END_VAR
VAR
	nPayloadRcvLen 			: UDINT;
END_VAR
STRNCPY( ADR(sMqttData.stTopic), ADR(topic), SIZEOF(sMqttData.stTopic) );
MEMSET(ADR(sMqttData.stMessage), 0, SIZEOF(sMqttData.stMessage));
FC_MemcpyLimited(ADR(sMqttData.stMessage), SIZEOF(sMqttData.stMessage), payload, length);

IF sMqttData.stTopic = 'shellyplus1pm-e465b8944d64/status/switch:0' THEN
	IF ParseStatusMessage(sMqttData.stMessage) = 'on' THEN
		sStatusDevices.sLivingRoom.sShellyLight.iOutput := 1;
	ELSIF ParseStatusMessage(sMqttData.stMessage) = 'off' THEN
		sStatusDevices.sLivingRoom.sShellyLight.iOutput := 0;
	END_IF
END_IF
END_METHOD

METHOD ParseStatusMessage : STRING(255)
VAR_INPUT
	istrMessage									: STRING(255);
END_VAR
VAR_OUTPUT	
END_VAR
VAR
	lstrMessage									: STRING(255);
	lstrTemp									: STRING(255);
	lxStringFound								: UDINT;
END_VAR
ParseStatusMessage := 'empty';
lstrMessage := istrMessage;

lstrTemp := 'true';
lxStringFound := FIND2(pSrcString:= ADR(lstrMessage), pFindString:= ADR(lstrTemp));
IF (lxStringFound > 0) THEN
	ParseStatusMessage := 'on';
	RETURN;
END_IF

lstrTemp := 'false';
lxStringFound := FIND2(pSrcString:= ADR(lstrMessage), pFindString:= ADR(lstrTemp));
IF (lxStringFound > 0) THEN
	ParseStatusMessage := 'off';
	RETURN;
END_IF
END_METHOD

END_FUNCTION_BLOCK
